// TIA Portal V15.1 export
// export: Created 2024-06-21T08:41:06.8182544Z, ExportSetting WithDefaults, DisplayName Totally Integrated Automation Portal, DisplayVersion V15.1 Update 5, DisplayName TIA Portal Openness, DisplayVersion V15.1 Update 5, DisplayName SINAMICS Startdrive Advanced, DisplayVersion V15.1, DisplayName G130, G150, S120, S150, SINAMICS MV, S210, DisplayVersion V15.1, DisplayName G110M, G120, G120C, G120D, G120P, DisplayVersion V15.1, DisplayName STEP 7 Professional, DisplayVersion V15.1 Update 5, DisplayName STEP 7 Safety, DisplayVersion V15.1, DisplayName WinCC Professional, DisplayVersion V15.1 Update 5, DisplayName SIMATIC Visualization Architect, DisplayVersion V15.1
FUNCTION_BLOCK "LGBProdStartStop"   // FB6645, FBD
TITLE = LGBProdStartStop
{ S7_Optimized_Access := 'TRUE' }
VERSION : 0.1
// stored: AutoNumber false, IsIECCheckEnabled false, IsRetainMemResEnabled false, MemoryReserve 100, SetENOAutomatically False, UDAEnableTagReadback false
   VAR_INPUT
      I_StartReqCR { ExternalAccessible := 'False'; ExternalVisible := 'False'; ExternalWritable := 'False'} : Bool;   // start request by controlroom
      I_StopReqCR { ExternalAccessible := 'False'; ExternalVisible := 'False'; ExternalWritable := 'False'} : Bool;   // stop request by controlroom
      I_StartReqPbLocal { ExternalAccessible := 'False'; ExternalVisible := 'False'; ExternalWritable := 'False'} : Bool;   // start request by local Pushbutton
      I_StopReqPbLocal { ExternalAccessible := 'False'; ExternalVisible := 'False'; ExternalWritable := 'False'} : Bool;   // stop request by local Pushbutton
      I_StopReqInfdWait { ExternalAccessible := 'False'; ExternalVisible := 'False'; ExternalWritable := 'False'} : Bool;   // stop request by infeed Wait state
      I_StopReqOutfdWait { ExternalAccessible := 'False'; ExternalVisible := 'False'; ExternalWritable := 'False'} : Bool;   // stop request by outfeed Wait state
      I_StopReqAndonHcall { ExternalAccessible := 'False'; ExternalVisible := 'False'; ExternalWritable := 'False'} : Bool;   // stop request by Andon - cause H call
      I_StopReqAndonEcall { ExternalAccessible := 'False'; ExternalVisible := 'False'; ExternalWritable := 'False'} : Bool;   // stop request by Andon - cause E call
      I_StopReqAndonMcall { ExternalAccessible := 'False'; ExternalVisible := 'False'; ExternalWritable := 'False'} : Bool;   // stop request by Andon - cause E call
      I_PartsAtFixedLineStop { ExternalAccessible := 'False'; ExternalVisible := 'False'; ExternalWritable := 'False'} : Bool;   // parts are at fixed linstop position (from linefeed module)
      I_SetpCycleTime { ExternalAccessible := 'False'; ExternalVisible := 'False'; ExternalWritable := 'False'} : Int := 60;   // Cycle time (s)
   END_VAR
   VAR_OUTPUT
      O_StartCmd { ExternalAccessible := 'False'; ExternalVisible := 'False'; ExternalWritable := 'False'} : Bool;   // start command to external unit
      O_StopCmd { ExternalAccessible := 'False'; ExternalVisible := 'False'; ExternalWritable := 'False'} : Bool;   // stop command to external unit
      O_IndStart { ExternalAccessible := 'False'; ExternalVisible := 'False'; ExternalWritable := 'False'} : Bool;   // Indication Start for button
      O_IndStop { ExternalAccessible := 'False'; ExternalVisible := 'False'; ExternalWritable := 'False'} : Bool;   // Indication Stop for button
      O_AndonActive { ExternalAccessible := 'False'; ExternalVisible := 'False'; ExternalWritable := 'False'} : Bool;   // andon is active
      O_StoppedByCR { ExternalAccessible := 'False'; ExternalVisible := 'False'; ExternalWritable := 'False'} : Bool;   // state 'stopped by controlroom' is active
      O_StoppedByLocal { ExternalAccessible := 'False'; ExternalVisible := 'False'; ExternalWritable := 'False'} : Bool;   // state 'stopped by local operator action ' is active
      O_StoppedByInfeedWait { ExternalAccessible := 'False'; ExternalVisible := 'False'; ExternalWritable := 'False'} : Bool;   // state 'stopped by infeed wait ' is active
      O_StoppedByOutfeedWait { ExternalAccessible := 'False'; ExternalVisible := 'False'; ExternalWritable := 'False'} : Bool;   // state 'stopped by outfeed wait ' is active
      O_StoppedByAndonHcall { ExternalAccessible := 'False'; ExternalVisible := 'False'; ExternalWritable := 'False'} : Bool;   // stopped by andon H-call
      O_StoppedByAndonEcall { ExternalAccessible := 'False'; ExternalVisible := 'False'; ExternalWritable := 'False'} : Bool;   // stopped by andon E-call
      O_StoppedByAndonMcall { ExternalAccessible := 'False'; ExternalVisible := 'False'; ExternalWritable := 'False'} : Bool;   // stopped by andon E-call
      O_GapsAllowed { ExternalAccessible := 'False'; ExternalVisible := 'False'; ExternalWritable := 'False'} : Bool;   // Gaps Allowed
      O_AlarmABCondition { ExternalAccessible := 'False'; ExternalVisible := 'False'; ExternalWritable := 'False'} : Bool;   // Alarm AB Condition
      O_AlarmA { ExternalAccessible := 'False'; ExternalVisible := 'False'; ExternalWritable := 'False'} : Bool;   // Summation Alarm A of roller. / Alarm A
      O_AlarmB { ExternalAccessible := 'False'; ExternalVisible := 'False'; ExternalWritable := 'False'} : Bool;   // Summation Alarm B of roller. / Alarm B
      O_AlarmC { ExternalAccessible := 'False'; ExternalVisible := 'False'; ExternalWritable := 'False'} : Bool;   // Summation Alarm C of roller. / Alarm C
      O_AlarmD { ExternalAccessible := 'False'; ExternalVisible := 'False'; ExternalWritable := 'False'} : Bool;   // Summation Alarm D of roller. / Alarm D
      H_AlarmDWord { ExternalAccessible := 'False'; ExternalVisible := 'False'; ExternalWritable := 'False'} : DWord;   // Alarm Word
   END_VAR
   VAR_IN_OUT
      IO_Modes : "Modes";   // Modes
      IO_ShiftRegData : "ShiftRegData";   // Line data- from shiftregister
      H_HMI : "H_HMI";   // Animation
      H_GBProdStartStop : "H_GBProdStartStop";   // Animation
      C_Config : "ProdStartStopConfig";   // Config
   END_VAR
   VAR
      AD_StopCR { ExternalAccessible := 'False'; ExternalVisible := 'False'; ExternalWritable := 'False'} : Bool;   // Stop by Control Room
      AD_StopLocal { ExternalAccessible := 'False'; ExternalVisible := 'False'; ExternalWritable := 'False'} : Bool;   // Stop by local stop
      AD_StopAndonHCall { ExternalAccessible := 'False'; ExternalVisible := 'False'; ExternalWritable := 'False'} : Bool;   // Stop by Andon H Call
      AD_StopAndonECall { ExternalAccessible := 'False'; ExternalVisible := 'False'; ExternalWritable := 'False'} : Bool;   // Stop by Andon E Call
      AD_StopAndonMCall { ExternalAccessible := 'False'; ExternalVisible := 'False'; ExternalWritable := 'False'} : Bool;   // Stop by Andon M Call
      AD_AndonNotActive { ExternalAccessible := 'False'; ExternalVisible := 'False'; ExternalWritable := 'False'} : Bool;   // Andon not active
      AD_StopInfeedWait { ExternalAccessible := 'False'; ExternalVisible := 'False'; ExternalWritable := 'False'} : Bool;   // Stop by infeed wait
      AD_StopOutfeedWait { ExternalAccessible := 'False'; ExternalVisible := 'False'; ExternalWritable := 'False'} : Bool;   // Stop by outfeed wait
      AD_GapsAllowed { ExternalAccessible := 'False'; ExternalVisible := 'False'; ExternalWritable := 'False'} : Bool;   // Gaps Allowed
      AndonActive { ExternalAccessible := 'False'; ExternalVisible := 'False'; ExternalWritable := 'False'} : Bool;
      StartReqCRDelayed { ExternalAccessible := 'False'; ExternalVisible := 'False'; ExternalWritable := 'False'} : Bool;
      StopReqCRCond { ExternalAccessible := 'False'; ExternalVisible := 'False'; ExternalWritable := 'False'} : Bool;
      StopReqCRPls { ExternalAccessible := 'False'; ExternalVisible := 'False'; ExternalWritable := 'False'} : Bool;
      StopReqCREdg { ExternalAccessible := 'False'; ExternalVisible := 'False'; ExternalWritable := 'False'} : Bool;
      StopReqCR { ExternalAccessible := 'False'; ExternalVisible := 'False'; ExternalWritable := 'False'} : Bool;
      StopReqCRDelayed { ExternalAccessible := 'False'; ExternalVisible := 'False'; ExternalWritable := 'False'} : Bool;
      StopReqDelayTimerAct { ExternalAccessible := 'False'; ExternalVisible := 'False'; ExternalWritable := 'False'} : DInt;
      StartReqHMIPls { ExternalAccessible := 'False'; ExternalVisible := 'False'; ExternalWritable := 'False'} : Bool;
      StartReqCRPls { ExternalAccessible := 'False'; ExternalVisible := 'False'; ExternalWritable := 'False'} : Bool;
      StartReqCREdg { ExternalAccessible := 'False'; ExternalVisible := 'False'; ExternalWritable := 'False'} : Bool;
      StopReqHMI { ExternalAccessible := 'False'; ExternalVisible := 'False'; ExternalWritable := 'False'} : Bool;
      StopReqAndon { ExternalAccessible := 'False'; ExternalVisible := 'False'; ExternalWritable := 'False'} : Bool;
      StoppedPrepared { ExternalAccessible := 'False'; ExternalVisible := 'False'; ExternalWritable := 'False'} : Bool;
      StartedPrepared { ExternalAccessible := 'False'; ExternalVisible := 'False'; ExternalWritable := 'False'} : Bool;
      StartedPreparedEdge { ExternalAccessible := 'False'; ExternalVisible := 'False'; ExternalWritable := 'False'} : Bool;
      StoppedAtLineOfTime { ExternalAccessible := 'False'; ExternalVisible := 'False'; ExternalWritable := 'False'} : Bool;
      StartReqCRDelayTimerSetp { ExternalAccessible := 'False'; ExternalVisible := 'False'; ExternalWritable := 'False'} : DInt;
      StartReqCRDelayTimerAct { ExternalAccessible := 'False'; ExternalVisible := 'False'; ExternalWritable := 'False'} : DInt;
      StartReqCRDelayTimerActRemain { ExternalAccessible := 'False'; ExternalVisible := 'False'; ExternalWritable := 'False'} : DInt;
      StartReqCRDelayTimerActRemainS { ExternalAccessible := 'False'; ExternalVisible := 'False'; ExternalWritable := 'False'} : DInt;
      StopReqHMIPls { ExternalAccessible := 'False'; ExternalVisible := 'False'; ExternalWritable := 'False'} : Bool;
      StopAndonReqHMIPls { ExternalAccessible := 'False'; ExternalVisible := 'False'; ExternalWritable := 'False'} : Bool;
      StopReqLocalPBEdg { ExternalAccessible := 'False'; ExternalVisible := 'False'; ExternalWritable := 'False'} : Bool;
      StopReqLocalPBPls { ExternalAccessible := 'False'; ExternalVisible := 'False'; ExternalWritable := 'False'} : Bool;
      StartReqLocalPBEdg { ExternalAccessible := 'False'; ExternalVisible := 'False'; ExternalWritable := 'False'} : Bool;
      StartReqLocalPBPls { ExternalAccessible := 'False'; ExternalVisible := 'False'; ExternalWritable := 'False'} : Bool;
      StopReqLocal { ExternalAccessible := 'False'; ExternalVisible := 'False'; ExternalWritable := 'False'} : Bool;
      Stop { ExternalAccessible := 'False'; ExternalVisible := 'False'; ExternalWritable := 'False'} : Bool;
      StoppedbyAndonHCall { ExternalAccessible := 'False'; ExternalVisible := 'False'; ExternalWritable := 'False'} : Bool;
      StoppedbyAndonECall { ExternalAccessible := 'False'; ExternalVisible := 'False'; ExternalWritable := 'False'} : Bool;
      StoppedbyAndonMCall { ExternalAccessible := 'False'; ExternalVisible := 'False'; ExternalWritable := 'False'} : Bool;
   END_VAR
   VAR RETAIN
      GapsAllowed { ExternalAccessible := 'False'; ExternalVisible := 'False'; ExternalWritable := 'False'} : Bool;
   END_VAR
   VAR
      AlarmA { ExternalAccessible := 'False'; ExternalVisible := 'False'; ExternalWritable := 'False'} : Bool;   // Summation Alarm A of roller. / Alarm A
      AlarmB { ExternalAccessible := 'False'; ExternalVisible := 'False'; ExternalWritable := 'False'} : Bool;   // Summation Alarm B of roller. / Alarm B
      AlarmC { ExternalAccessible := 'False'; ExternalVisible := 'False'; ExternalWritable := 'False'} : Bool;   // Summation Alarm C of roller. / Alarm C
      AlarmD { ExternalAccessible := 'False'; ExternalVisible := 'False'; ExternalWritable := 'False'} : Bool;   // Summation Alarm D of roller. / Alarm D
      AlarmABCondition { ExternalAccessible := 'False'; ExternalVisible := 'False'; ExternalWritable := 'False'} : Bool;   // Alarm AB Condition
      CycleTimeSetp { ExternalAccessible := 'False'; ExternalVisible := 'False'; ExternalWritable := 'False'} : DInt;   // cycletime (ms)
      HMICMD { ExternalAccessible := 'False'; ExternalVisible := 'False'; ExternalWritable := 'False'} : Struct   // Temp
         Start { ExternalAccessible := 'False'; ExternalVisible := 'False'; ExternalWritable := 'False'} : Bool;   // Start
         Stop { ExternalAccessible := 'False'; ExternalVisible := 'False'; ExternalWritable := 'False'} : Bool;   // Stop
         StopAndon { ExternalAccessible := 'False'; ExternalVisible := 'False'; ExternalWritable := 'False'} : Bool;   // Stop Andon
         ActivateAndon { ExternalAccessible := 'False'; ExternalVisible := 'False'; ExternalWritable := 'False'} : Bool;   // Activate Andon
         GapsAllowed { ExternalAccessible := 'False'; ExternalVisible := 'False'; ExternalWritable := 'False'} : Bool;   // Gaps Allowed
         Spare5 { ExternalAccessible := 'False'; ExternalVisible := 'False'; ExternalWritable := 'False'} : Bool;   // Spare
         Spare6 { ExternalAccessible := 'False'; ExternalVisible := 'False'; ExternalWritable := 'False'} : Bool;   // Spare
         Spare7 { ExternalAccessible := 'False'; ExternalVisible := 'False'; ExternalWritable := 'False'} : Bool;   // Spare
         Spare8 { ExternalAccessible := 'False'; ExternalVisible := 'False'; ExternalWritable := 'False'} : Bool;   // Spare
         Spare9 { ExternalAccessible := 'False'; ExternalVisible := 'False'; ExternalWritable := 'False'} : Bool;   // Spare
         Spare10 { ExternalAccessible := 'False'; ExternalVisible := 'False'; ExternalWritable := 'False'} : Bool;   // Spare
         Spare11 { ExternalAccessible := 'False'; ExternalVisible := 'False'; ExternalWritable := 'False'} : Bool;   // Spare
         Spare12 { ExternalAccessible := 'False'; ExternalVisible := 'False'; ExternalWritable := 'False'} : Bool;   // Spare
         Spare13 { ExternalAccessible := 'False'; ExternalVisible := 'False'; ExternalWritable := 'False'} : Bool;   // Spare
         Spare14 { ExternalAccessible := 'False'; ExternalVisible := 'False'; ExternalWritable := 'False'} : Bool;   // Spare
         Spare15 { ExternalAccessible := 'False'; ExternalVisible := 'False'; ExternalWritable := 'False'} : Bool;   // Spare
         Spare16 { ExternalAccessible := 'False'; ExternalVisible := 'False'; ExternalWritable := 'False'} : Bool;   // Spare
         Spare17 { ExternalAccessible := 'False'; ExternalVisible := 'False'; ExternalWritable := 'False'} : Bool;   // Spare
         Spare18 { ExternalAccessible := 'False'; ExternalVisible := 'False'; ExternalWritable := 'False'} : Bool;   // Spare
         Spare19 { ExternalAccessible := 'False'; ExternalVisible := 'False'; ExternalWritable := 'False'} : Bool;   // Spare
         Spare20 { ExternalAccessible := 'False'; ExternalVisible := 'False'; ExternalWritable := 'False'} : Bool;   // Spare
         Spare21 { ExternalAccessible := 'False'; ExternalVisible := 'False'; ExternalWritable := 'False'} : Bool;   // Spare
         Spare22 { ExternalAccessible := 'False'; ExternalVisible := 'False'; ExternalWritable := 'False'} : Bool;   // Spare
         Spare23 { ExternalAccessible := 'False'; ExternalVisible := 'False'; ExternalWritable := 'False'} : Bool;   // Spare
         Spare24 { ExternalAccessible := 'False'; ExternalVisible := 'False'; ExternalWritable := 'False'} : Bool;   // Spare
         Spare25 { ExternalAccessible := 'False'; ExternalVisible := 'False'; ExternalWritable := 'False'} : Bool;   // Spare
         Spare26 { ExternalAccessible := 'False'; ExternalVisible := 'False'; ExternalWritable := 'False'} : Bool;   // Spare
         Spare27 { ExternalAccessible := 'False'; ExternalVisible := 'False'; ExternalWritable := 'False'} : Bool;   // Spare
         Spare28 { ExternalAccessible := 'False'; ExternalVisible := 'False'; ExternalWritable := 'False'} : Bool;   // Spare
         Spare29 { ExternalAccessible := 'False'; ExternalVisible := 'False'; ExternalWritable := 'False'} : Bool;   // Spare
         Spare30 { ExternalAccessible := 'False'; ExternalVisible := 'False'; ExternalWritable := 'False'} : Bool;   // Spare
         Spare31 { ExternalAccessible := 'False'; ExternalVisible := 'False'; ExternalWritable := 'False'} : Bool;   // Spare
      END_STRUCT;
      _StartReqCRDelayTimer { ExternalAccessible := 'False'; ExternalVisible := 'False'; ExternalWritable := 'False'} : "LTimer";
      _StopReqCRDelayTimer { ExternalAccessible := 'False'; ExternalVisible := 'False'; ExternalWritable := 'False'} : "LTimer";
      LToggle_GapsAllowed { ExternalAccessible := 'False'; ExternalVisible := 'False'; ExternalWritable := 'False'} : "LToggle";
   END_VAR
   VAR_TEMP   // added for the SCL form of the ladder/FBD networks
      _w1 : Bool;
      _w2 : Bool;
   END_VAR
BEGIN

REGION Network 1: **** 1 - Inputs **** HMI Commands
   // HMI Commands
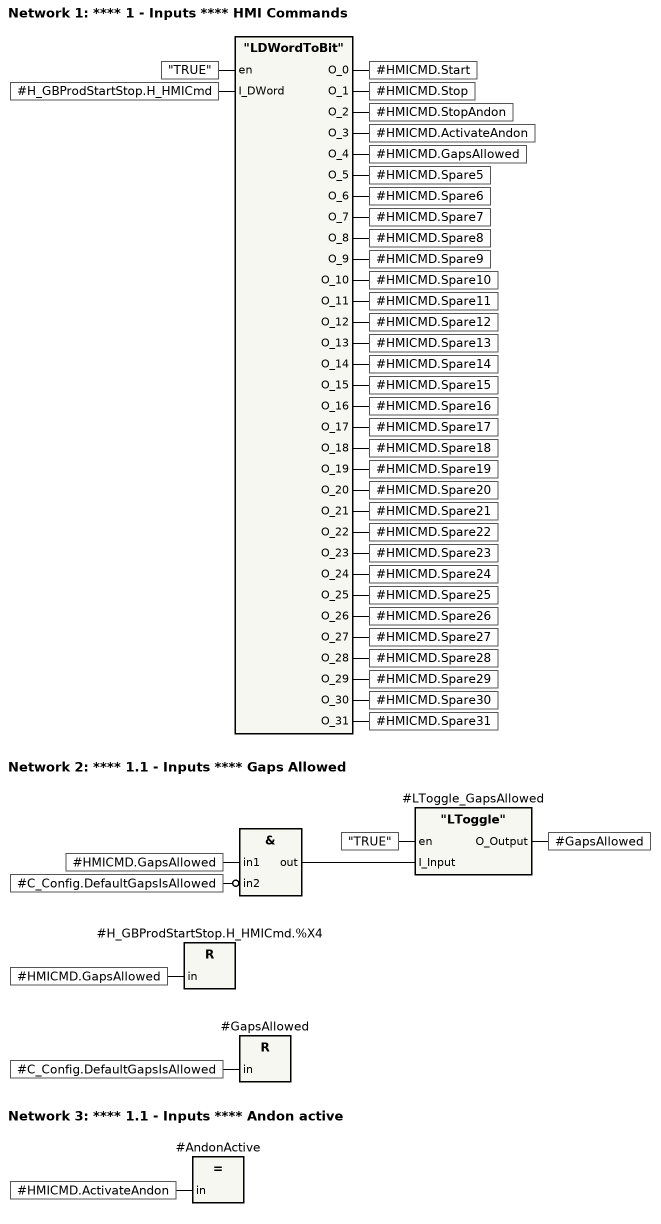
   IF "TRUE" THEN
       "LDWordToBit"(I_DWord := #H_GBProdStartStop.H_HMICmd,
                     O_0 => #HMICMD.Start,
                     O_1 => #HMICMD.Stop,
                     O_2 => #HMICMD.StopAndon,
                     O_3 => #HMICMD.ActivateAndon,
                     O_4 => #HMICMD.GapsAllowed,
                     O_5 => #HMICMD.Spare5,
                     O_6 => #HMICMD.Spare6,
                     O_7 => #HMICMD.Spare7,
                     O_8 => #HMICMD.Spare8,
                     O_9 => #HMICMD.Spare9,
                     O_10 => #HMICMD.Spare10,
                     O_11 => #HMICMD.Spare11,
                     O_12 => #HMICMD.Spare12,
                     O_13 => #HMICMD.Spare13,
                     O_14 => #HMICMD.Spare14,
                     O_15 => #HMICMD.Spare15,
                     O_16 => #HMICMD.Spare16,
                     O_17 => #HMICMD.Spare17,
                     O_18 => #HMICMD.Spare18,
                     O_19 => #HMICMD.Spare19,
                     O_20 => #HMICMD.Spare20,
                     O_21 => #HMICMD.Spare21,
                     O_22 => #HMICMD.Spare22,
                     O_23 => #HMICMD.Spare23,
                     O_24 => #HMICMD.Spare24,
                     O_25 => #HMICMD.Spare25,
                     O_26 => #HMICMD.Spare26,
                     O_27 => #HMICMD.Spare27,
                     O_28 => #HMICMD.Spare28,
                     O_29 => #HMICMD.Spare29,
                     O_30 => #HMICMD.Spare30,
                     O_31 => #HMICMD.Spare31);
   END_IF;
END_REGION

REGION Network 2: **** 1.1 - Inputs **** Gaps Allowed
   IF "TRUE" THEN
       #LToggle_GapsAllowed(I_Input := #HMICMD.GapsAllowed AND NOT #C_Config.DefaultGapsIsAllowed,   // "LToggle"
                            O_Output => #GapsAllowed);
   END_IF;
   IF #HMICMD.GapsAllowed THEN #H_GBProdStartStop.H_HMICmd.%X4 := FALSE; END_IF;
   IF #C_Config.DefaultGapsIsAllowed THEN #GapsAllowed := FALSE; END_IF;
END_REGION

REGION Network 3: **** 1.1 - Inputs **** Andon active
   #AndonActive := #HMICMD.ActivateAndon;
END_REGION

REGION Network 4: **** 1.1 - Inputs **** Pushbutton start request - by HMI - Create pulse
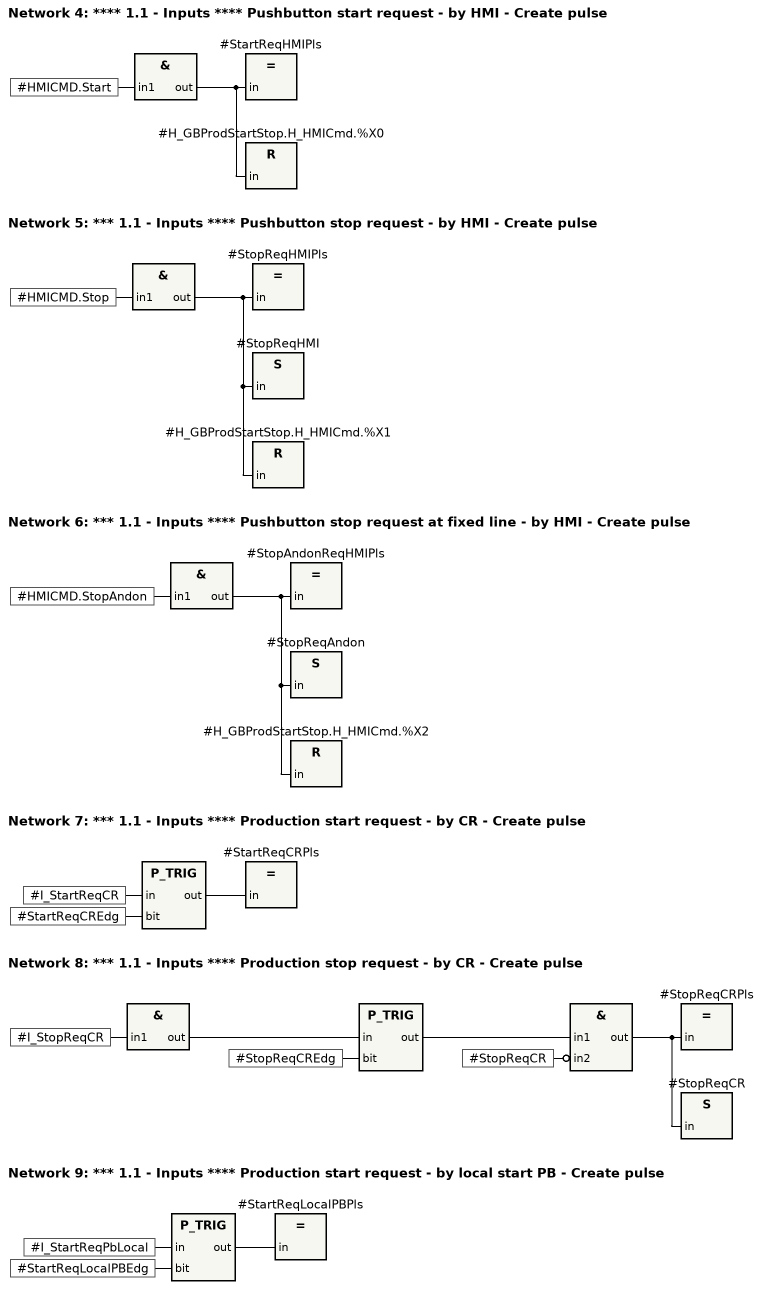
   #StartReqHMIPls := #HMICMD.Start;
   IF #HMICMD.Start THEN #H_GBProdStartStop.H_HMICmd.%X0 := FALSE; END_IF;
END_REGION

REGION Network 5: *** 1.1 - Inputs **** Pushbutton stop request - by HMI - Create pulse
   #StopReqHMIPls := #HMICMD.Stop;
   IF #HMICMD.Stop THEN
       #StopReqHMI := TRUE;
       #H_GBProdStartStop.H_HMICmd.%X1 := FALSE;
   END_IF;
END_REGION

REGION Network 6: *** 1.1 - Inputs **** Pushbutton stop request at fixed line - by HMI - Create pulse
   #StopAndonReqHMIPls := #HMICMD.StopAndon;
   IF #HMICMD.StopAndon THEN
       #StopReqAndon := TRUE;
       #H_GBProdStartStop.H_HMICmd.%X2 := FALSE;
   END_IF;
END_REGION

REGION Network 7: *** 1.1 - Inputs **** Production start request - by CR - Create pulse
   #_w1 := #I_StartReqCR AND NOT #StartReqCREdg;   // rising edge
   #StartReqCREdg := #I_StartReqCR;
   #StartReqCRPls := #_w1;
END_REGION

REGION Network 8: *** 1.1 - Inputs **** Production stop request - by CR - Create pulse
   #_w1 := #I_StopReqCR AND NOT #StopReqCREdg;   // rising edge
   #StopReqCREdg := #I_StopReqCR;
   #StopReqCRPls := #_w1 AND NOT #StopReqCR;
   IF #StopReqCRPls THEN #StopReqCR := TRUE; END_IF;
END_REGION

REGION Network 9: *** 1.1 - Inputs **** Production start request - by local start PB - Create pulse
   #_w1 := #I_StartReqPbLocal AND NOT #StartReqLocalPBEdg;   // rising edge
   #StartReqLocalPBEdg := #I_StartReqPbLocal;
   #StartReqLocalPBPls := #_w1;
END_REGION

REGION Network 10: *** 1.1 - Inputs **** Production stop request - by local stop PB - Create pulse
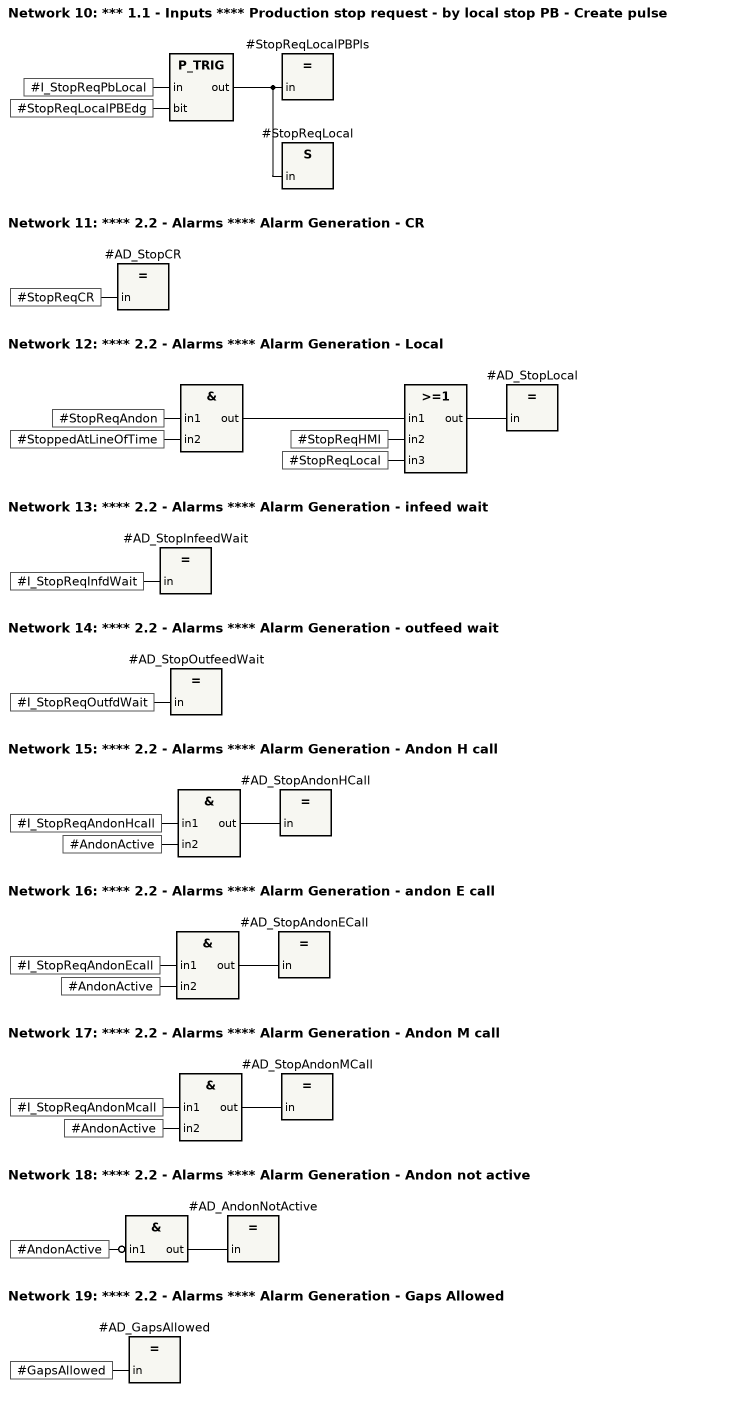
   #_w1 := #I_StopReqPbLocal AND NOT #StopReqLocalPBEdg;   // rising edge
   #StopReqLocalPBEdg := #I_StopReqPbLocal;
   #StopReqLocalPBPls := #_w1;
   IF #_w1 THEN #StopReqLocal := TRUE; END_IF;
END_REGION

REGION Network 11: **** 2.2 - Alarms **** Alarm Generation - CR
   #AD_StopCR := #StopReqCR;
END_REGION

REGION Network 12: **** 2.2 - Alarms **** Alarm Generation - Local
   #AD_StopLocal := (#StopReqAndon AND #StoppedAtLineOfTime) OR #StopReqHMI OR #StopReqLocal;
END_REGION

REGION Network 13: **** 2.2 - Alarms **** Alarm Generation - infeed wait
   #AD_StopInfeedWait := #I_StopReqInfdWait;
END_REGION

REGION Network 14: **** 2.2 - Alarms **** Alarm Generation - outfeed wait
   #AD_StopOutfeedWait := #I_StopReqOutfdWait;
END_REGION

REGION Network 15: **** 2.2 - Alarms **** Alarm Generation - Andon H call
   #AD_StopAndonHCall := #I_StopReqAndonHcall AND #AndonActive;
END_REGION

REGION Network 16: **** 2.2 - Alarms **** Alarm Generation - andon E call
   #AD_StopAndonECall := #I_StopReqAndonEcall AND #AndonActive;
END_REGION

REGION Network 17: **** 2.2 - Alarms **** Alarm Generation - Andon M call
   #AD_StopAndonMCall := #I_StopReqAndonMcall AND #AndonActive;
END_REGION

REGION Network 18: **** 2.2 - Alarms **** Alarm Generation - Andon not active
   #AD_AndonNotActive := NOT #AndonActive;
END_REGION

REGION Network 19: **** 2.2 - Alarms **** Alarm Generation - Gaps Allowed
   #AD_GapsAllowed := #GapsAllowed;
END_REGION

REGION Network 20: *** 4.6 - Machine Status - Indication **** Icon Animation
   // Icon Animation
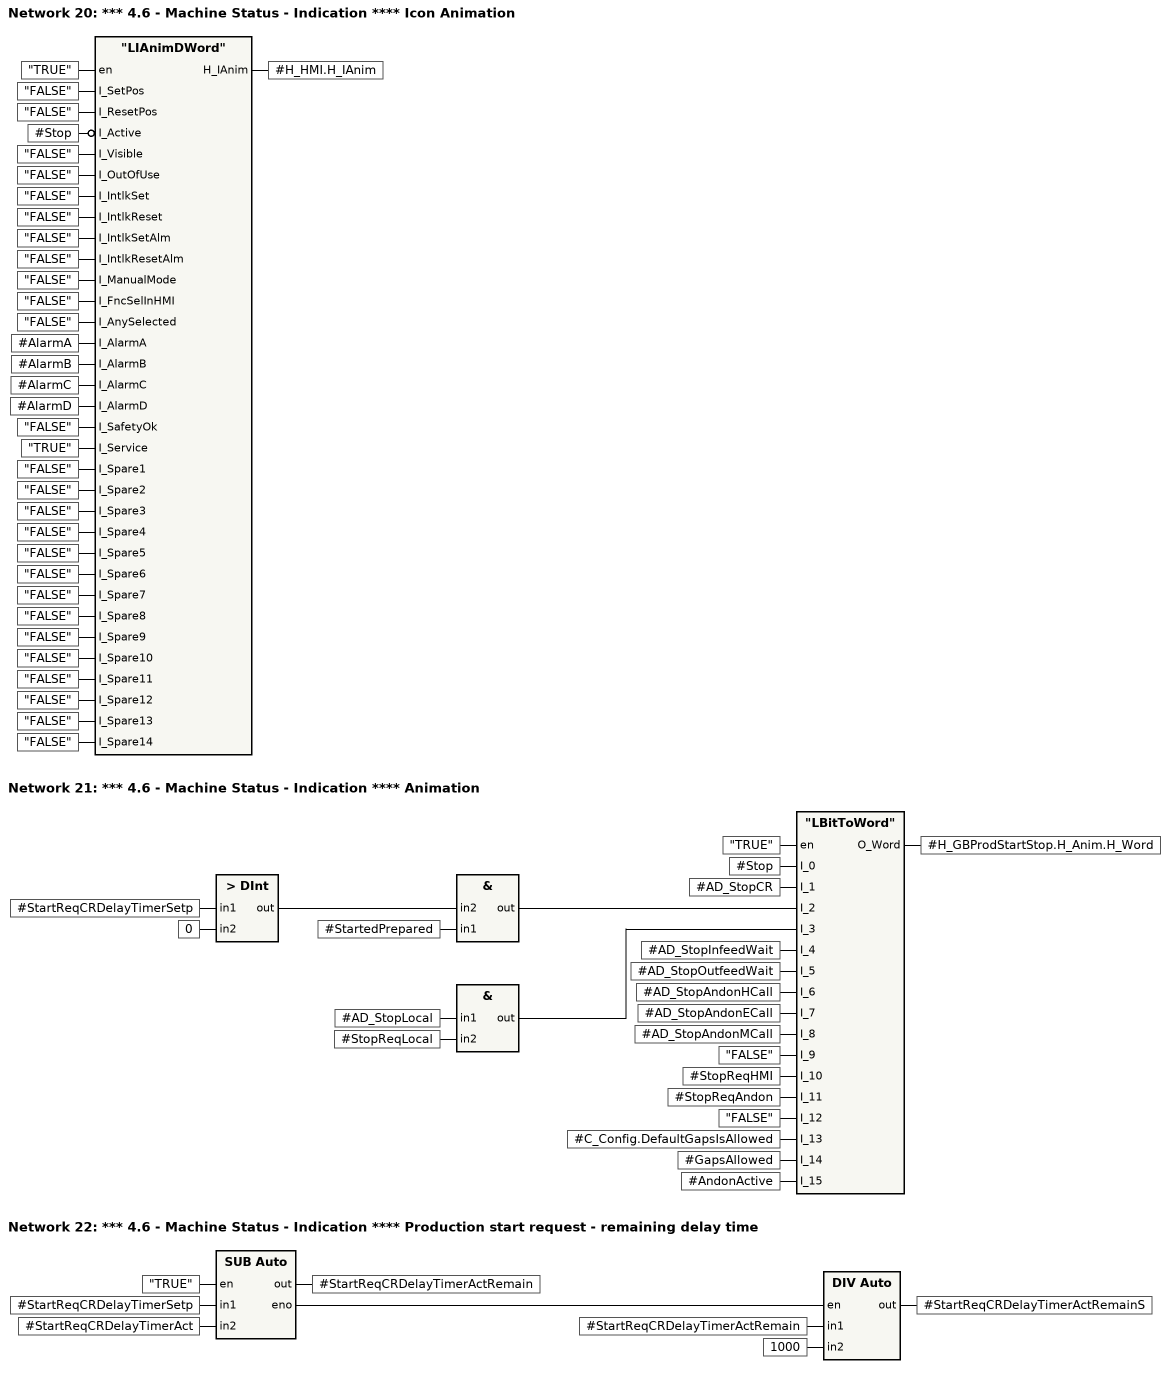
   IF "TRUE" THEN
       "LIAnimDWord"(I_SetPos := "FALSE",
                     I_ResetPos := "FALSE",
                     I_Active := NOT #Stop,
                     I_Visible := "FALSE",
                     I_OutOfUse := "FALSE",
                     I_IntlkSet := "FALSE",
                     I_IntlkReset := "FALSE",
                     I_IntlkSetAlm := "FALSE",
                     I_IntlkResetAlm := "FALSE",
                     I_ManualMode := "FALSE",
                     I_FncSelInHMI := "FALSE",
                     I_AnySelected := "FALSE",
                     I_AlarmA := #AlarmA,
                     I_AlarmB := #AlarmB,
                     I_AlarmC := #AlarmC,
                     I_AlarmD := #AlarmD,
                     I_SafetyOk := "FALSE",
                     I_Service := "TRUE",
                     I_Spare1 := "FALSE",
                     I_Spare2 := "FALSE",
                     I_Spare3 := "FALSE",
                     I_Spare4 := "FALSE",
                     I_Spare5 := "FALSE",
                     I_Spare6 := "FALSE",
                     I_Spare7 := "FALSE",
                     I_Spare8 := "FALSE",
                     I_Spare9 := "FALSE",
                     I_Spare10 := "FALSE",
                     I_Spare11 := "FALSE",
                     I_Spare12 := "FALSE",
                     I_Spare13 := "FALSE",
                     I_Spare14 := "FALSE",
                     H_IAnim => #H_HMI.H_IAnim);
   END_IF;
END_REGION

REGION Network 21: *** 4.6 - Machine Status - Indication **** Animation
   IF "TRUE" THEN
       "LBitToWord"(I_0 := #Stop,
                    I_1 := #AD_StopCR,
                    I_2 := (#StartReqCRDelayTimerSetp > 0) AND #StartedPrepared,
                    I_3 := #AD_StopLocal AND #StopReqLocal,
                    I_4 := #AD_StopInfeedWait,
                    I_5 := #AD_StopOutfeedWait,
                    I_6 := #AD_StopAndonHCall,
                    I_7 := #AD_StopAndonECall,
                    I_8 := #AD_StopAndonMCall,
                    I_9 := "FALSE",
                    I_10 := #StopReqHMI,
                    I_11 := #StopReqAndon,
                    I_12 := "FALSE",
                    I_13 := #C_Config.DefaultGapsIsAllowed,
                    I_14 := #GapsAllowed,
                    I_15 := #AndonActive,
                    O_Word => #H_GBProdStartStop.H_Anim.H_Word);
   END_IF;
END_REGION

REGION Network 22: *** 4.6 - Machine Status - Indication **** Production start request - remaining delay time
   IF "TRUE" THEN
       #StartReqCRDelayTimerActRemain := #StartReqCRDelayTimerSetp - #StartReqCRDelayTimerAct;
       #StartReqCRDelayTimerActRemainS := #StartReqCRDelayTimerActRemain / 1000;
   END_IF;
END_REGION

REGION Network 23: *** 4.6 - Machine Status - Indication **** Wait time start
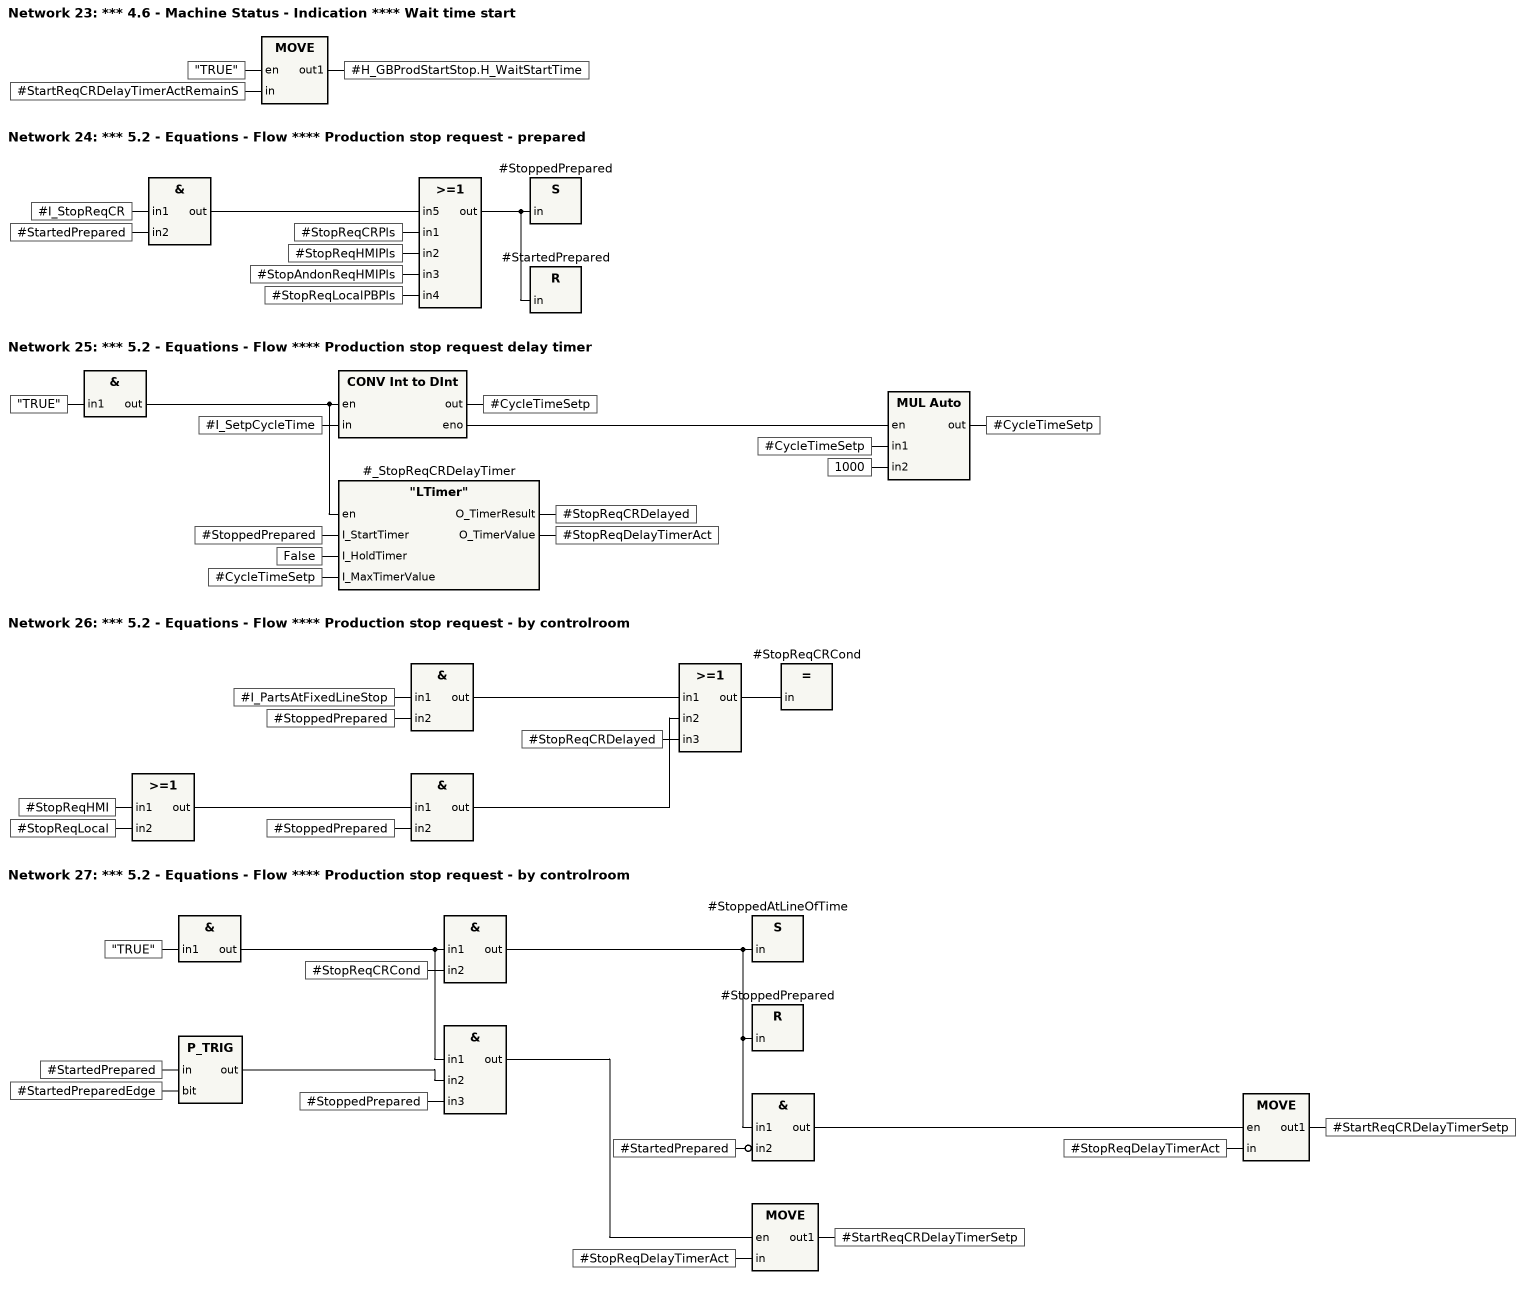
   IF "TRUE" THEN #H_GBProdStartStop.H_WaitStartTime := #StartReqCRDelayTimerActRemainS; END_IF;
END_REGION

REGION Network 24: *** 5.2 - Equations - Flow **** Production stop request - prepared
   IF (#I_StopReqCR AND #StartedPrepared) OR #StopReqCRPls OR #StopReqHMIPls OR #StopAndonReqHMIPls OR #StopReqLocalPBPls THEN
       #StoppedPrepared := TRUE;
       #StartedPrepared := FALSE;
   END_IF;
END_REGION

REGION Network 25: *** 5.2 - Equations - Flow **** Production stop request delay timer
   IF "TRUE" THEN
       #CycleTimeSetp := INT_TO_DINT(#I_SetpCycleTime);
       #CycleTimeSetp := #CycleTimeSetp * 1000;
       #_StopReqCRDelayTimer(I_StartTimer := #StoppedPrepared,   // "LTimer"
                             I_HoldTimer := False,
                             I_MaxTimerValue := #CycleTimeSetp,
                             O_TimerResult => #StopReqCRDelayed,
                             O_TimerValue => #StopReqDelayTimerAct);
   END_IF;
END_REGION

REGION Network 26: *** 5.2 - Equations - Flow **** Production stop request - by controlroom
   #StopReqCRCond := (#I_PartsAtFixedLineStop AND #StoppedPrepared) OR ((#StopReqHMI OR #StopReqLocal) AND #StoppedPrepared) OR #StopReqCRDelayed;
END_REGION

REGION Network 27: *** 5.2 - Equations - Flow **** Production stop request - by controlroom
   #_w1 := "TRUE" AND #StopReqCRCond;
   IF #_w1 THEN
       #StoppedAtLineOfTime := TRUE;
       #StoppedPrepared := FALSE;
   END_IF;
   IF #_w1 AND NOT #StartedPrepared THEN #StartReqCRDelayTimerSetp := #StopReqDelayTimerAct; END_IF;
   #_w2 := #StartedPrepared AND NOT #StartedPreparedEdge;   // rising edge
   #StartedPreparedEdge := #StartedPrepared;
   IF "TRUE" AND #_w2 AND #StoppedPrepared THEN #StartReqCRDelayTimerSetp := #StopReqDelayTimerAct; END_IF;
END_REGION

REGION Network 28: *** 5.2 - Equations - Flow **** Production start request - prepared
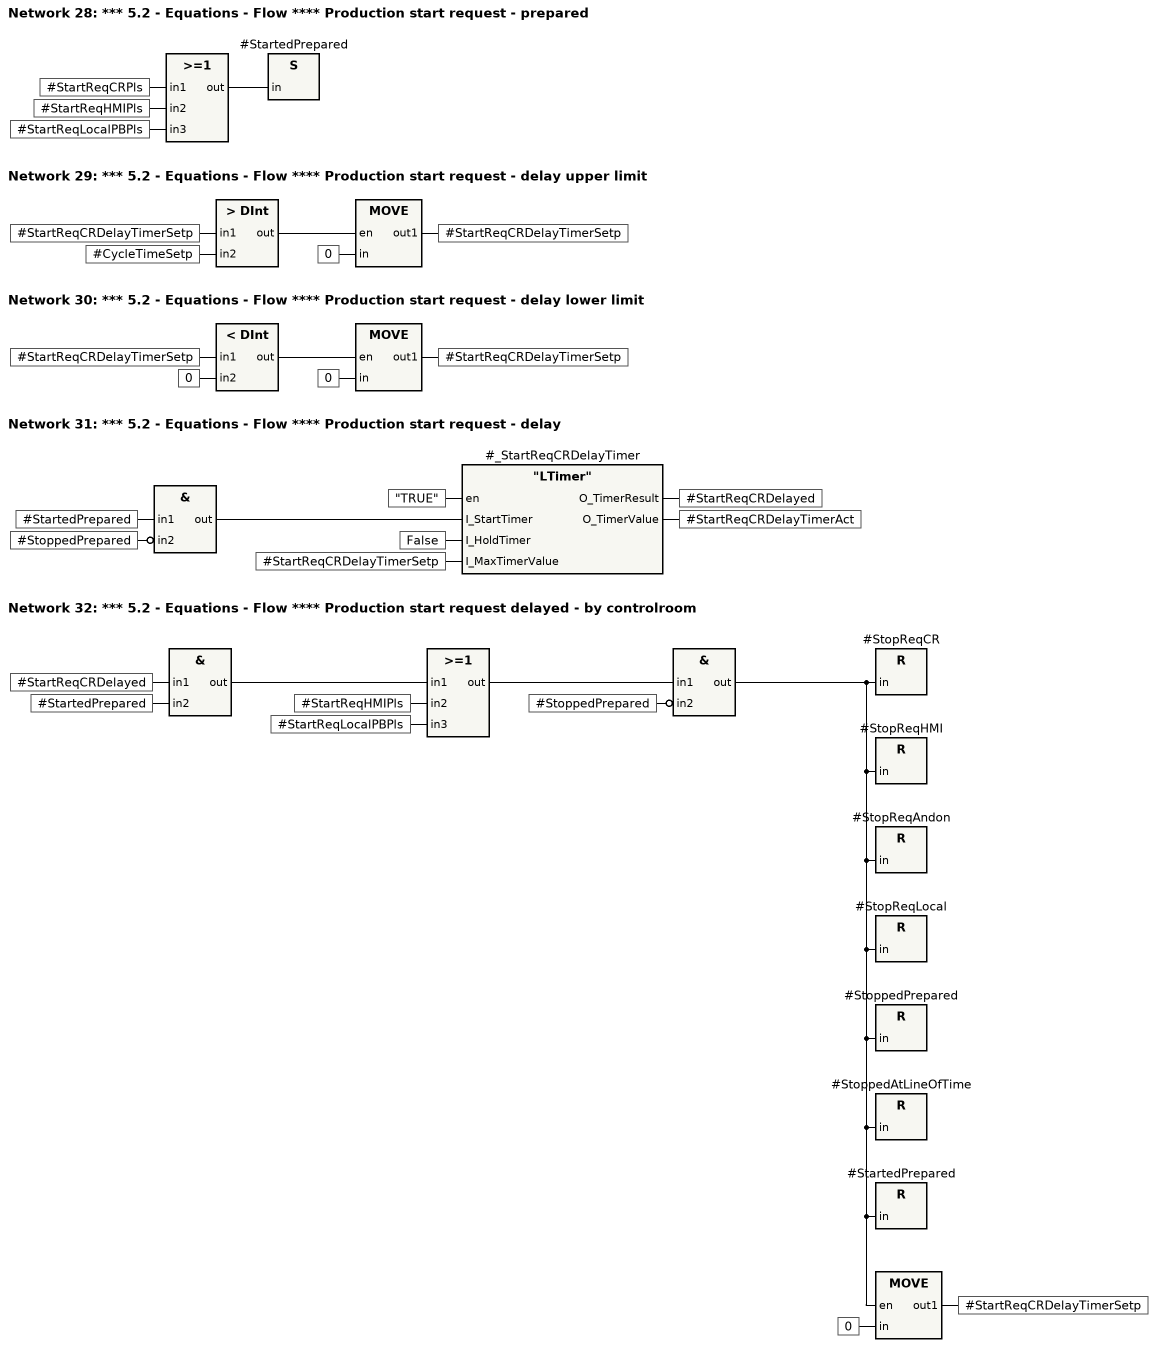
   IF #StartReqCRPls OR #StartReqHMIPls OR #StartReqLocalPBPls THEN #StartedPrepared := TRUE; END_IF;
END_REGION

REGION Network 29: *** 5.2 - Equations - Flow **** Production start request - delay upper limit
   IF #StartReqCRDelayTimerSetp > #CycleTimeSetp THEN #StartReqCRDelayTimerSetp := 0; END_IF;
END_REGION

REGION Network 30: *** 5.2 - Equations - Flow **** Production start request - delay lower limit
   IF #StartReqCRDelayTimerSetp < 0 THEN #StartReqCRDelayTimerSetp := 0; END_IF;
END_REGION

REGION Network 31: *** 5.2 - Equations - Flow **** Production start request - delay
   IF "TRUE" THEN
       #_StartReqCRDelayTimer(I_StartTimer := #StartedPrepared AND NOT #StoppedPrepared,   // "LTimer"
                              I_HoldTimer := False,
                              I_MaxTimerValue := #StartReqCRDelayTimerSetp,
                              O_TimerResult => #StartReqCRDelayed,
                              O_TimerValue => #StartReqCRDelayTimerAct);
   END_IF;
END_REGION

REGION Network 32: *** 5.2 - Equations - Flow **** Production start request delayed - by controlroom
   IF ((#StartReqCRDelayed AND #StartedPrepared) OR #StartReqHMIPls OR #StartReqLocalPBPls) AND NOT #StoppedPrepared THEN
       #StopReqCR := FALSE;
       #StopReqHMI := FALSE;
       #StopReqAndon := FALSE;
       #StopReqLocal := FALSE;
   END_IF;
   #_w1 := ((#StartReqCRDelayed AND #StartedPrepared) OR #StartReqHMIPls OR #StartReqLocalPBPls) AND NOT #StoppedPrepared;
   IF #_w1 THEN
       #StoppedPrepared := FALSE;
       #StoppedAtLineOfTime := FALSE;
       #StartedPrepared := FALSE;
       #StartReqCRDelayTimerSetp := 0;
   END_IF;
END_REGION

REGION Network 33: *** 5.2 - Equations - Flow **** stopped at line of time
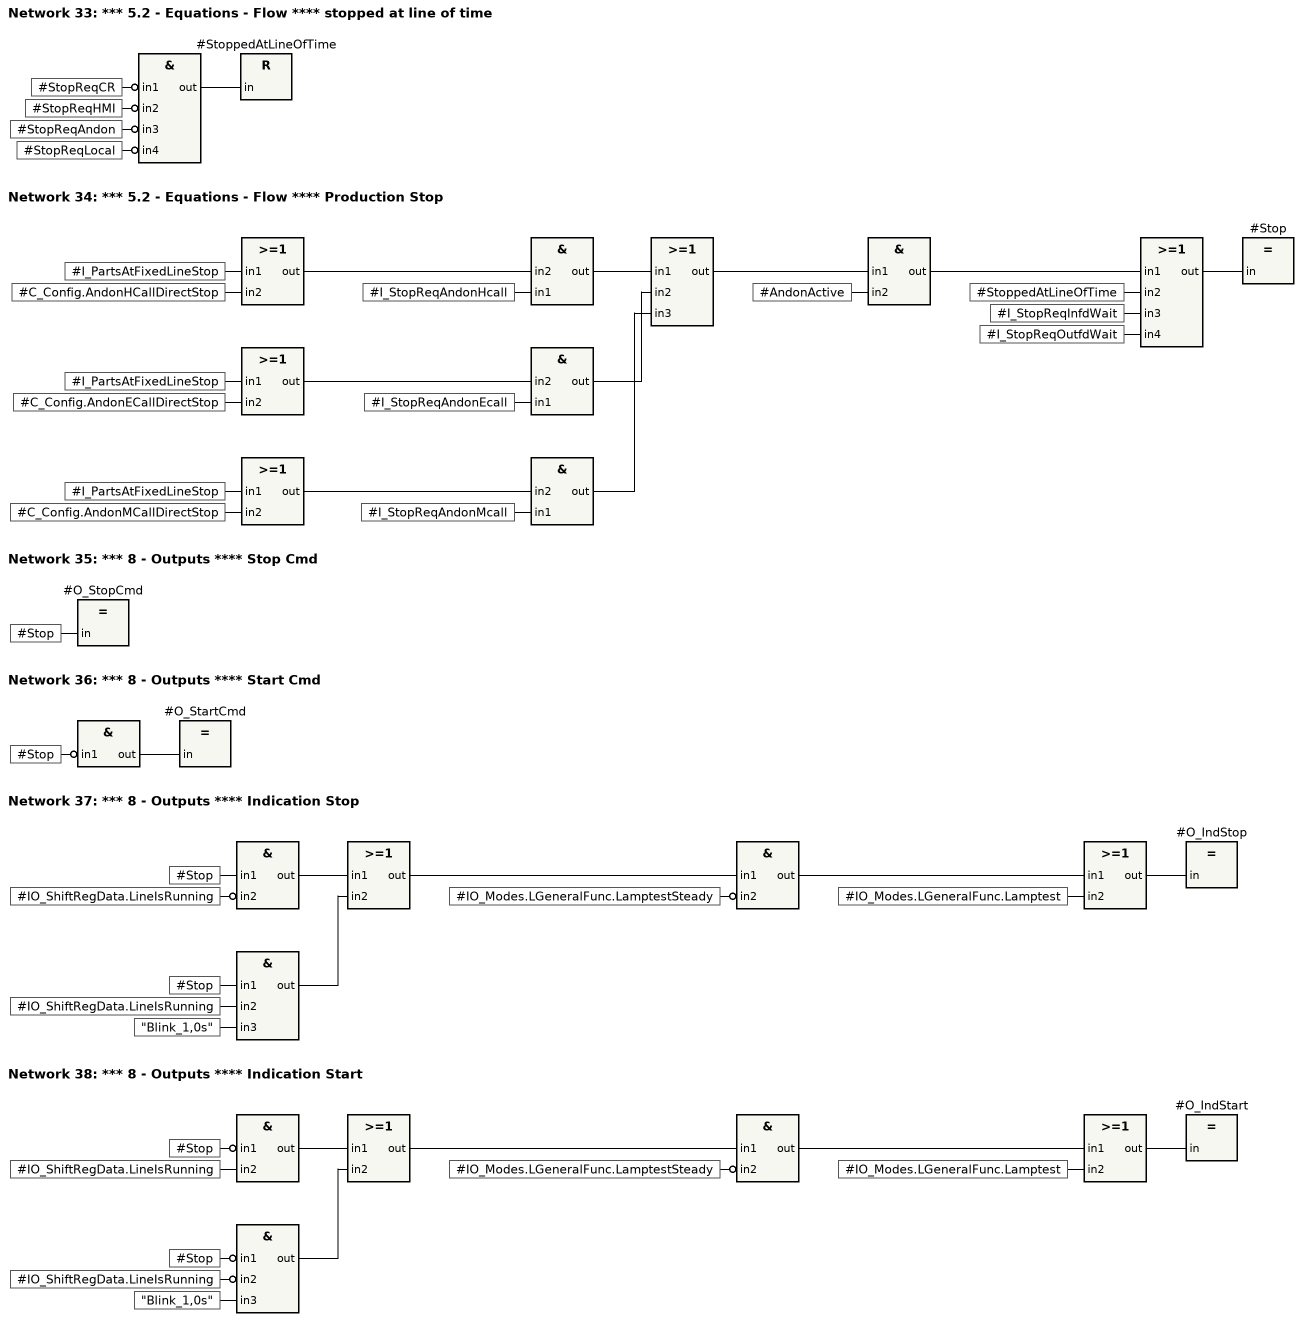
   IF NOT #StopReqCR AND NOT #StopReqHMI AND NOT #StopReqAndon AND NOT #StopReqLocal THEN
       #StoppedAtLineOfTime := FALSE;
   END_IF;
END_REGION

REGION Network 34: *** 5.2 - Equations - Flow **** Production Stop
   #Stop := ((((#I_PartsAtFixedLineStop OR #C_Config.AndonHCallDirectStop) AND #I_StopReqAndonHcall) OR ((#I_PartsAtFixedLineStop OR #C_Config.AndonECallDirectStop) AND #I_StopReqAndonEcall) OR ((#I_PartsAtFixedLineStop OR #C_Config.AndonMCallDirectStop) AND #I_StopReqAndonMcall)) AND #AndonActive) OR #StoppedAtLineOfTime OR #I_StopReqInfdWait OR #I_StopReqOutfdWait;
END_REGION

REGION Network 35: *** 8 - Outputs **** Stop Cmd
   #O_StopCmd := #Stop;
END_REGION

REGION Network 36: *** 8 - Outputs **** Start Cmd
   #O_StartCmd := NOT #Stop;
END_REGION

REGION Network 37: *** 8 - Outputs **** Indication Stop
   #O_IndStop := (((#Stop AND NOT #IO_ShiftRegData.LineIsRunning) OR (#Stop AND #IO_ShiftRegData.LineIsRunning AND "Blink_1,0s")) AND NOT #IO_Modes.LGeneralFunc.LamptestSteady) OR #IO_Modes.LGeneralFunc.Lamptest;
END_REGION

REGION Network 38: *** 8 - Outputs **** Indication Start
   #O_IndStart := (((NOT #Stop AND #IO_ShiftRegData.LineIsRunning) OR (NOT #Stop AND NOT #IO_ShiftRegData.LineIsRunning AND "Blink_1,0s")) AND NOT #IO_Modes.LGeneralFunc.LamptestSteady) OR #IO_Modes.LGeneralFunc.Lamptest;
END_REGION

REGION Network 39: *** 8 - Outputs **** Andon active
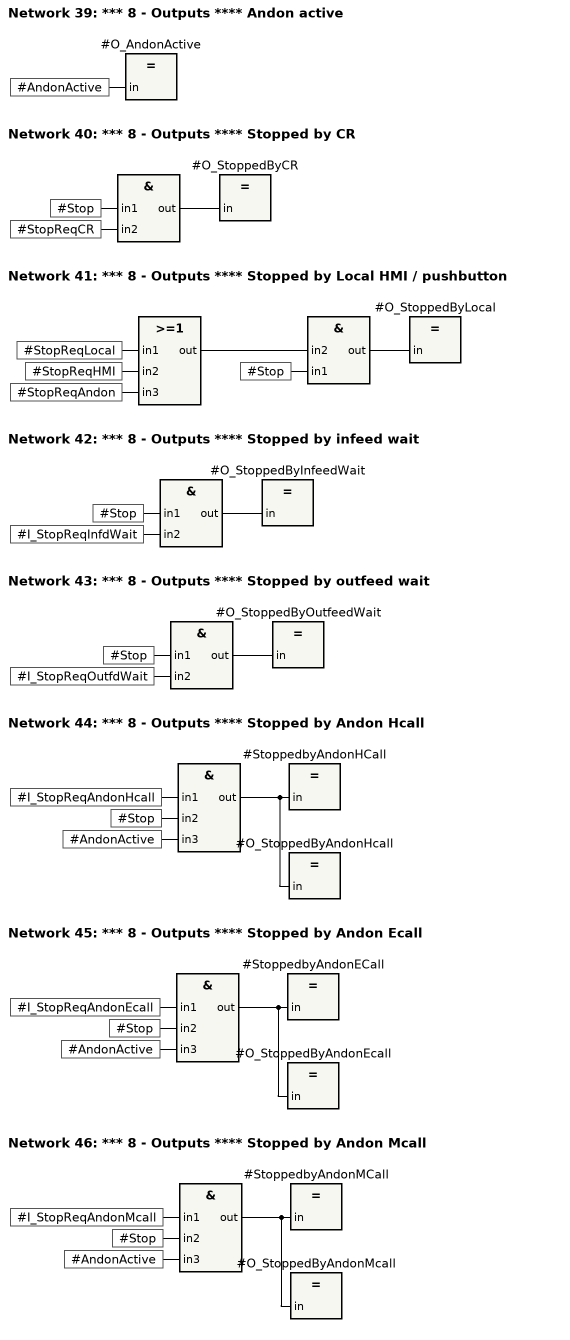
   #O_AndonActive := #AndonActive;
END_REGION

REGION Network 40: *** 8 - Outputs **** Stopped by CR
   #O_StoppedByCR := #Stop AND #StopReqCR;
END_REGION

REGION Network 41: *** 8 - Outputs **** Stopped by Local HMI / pushbutton
   #O_StoppedByLocal := (#StopReqLocal OR #StopReqHMI OR #StopReqAndon) AND #Stop;
END_REGION

REGION Network 42: *** 8 - Outputs **** Stopped by infeed wait
   #O_StoppedByInfeedWait := #Stop AND #I_StopReqInfdWait;
END_REGION

REGION Network 43: *** 8 - Outputs **** Stopped by outfeed wait
   #O_StoppedByOutfeedWait := #Stop AND #I_StopReqOutfdWait;
END_REGION

REGION Network 44: *** 8 - Outputs **** Stopped by Andon Hcall
   #StoppedbyAndonHCall := #I_StopReqAndonHcall AND #Stop AND #AndonActive;
   #O_StoppedByAndonHcall := #StoppedbyAndonHCall;
END_REGION

REGION Network 45: *** 8 - Outputs **** Stopped by Andon Ecall
   #StoppedbyAndonECall := #I_StopReqAndonEcall AND #Stop AND #AndonActive;
   #O_StoppedByAndonEcall := #StoppedbyAndonECall;
END_REGION

REGION Network 46: *** 8 - Outputs **** Stopped by Andon Mcall
   #StoppedbyAndonMCall := #I_StopReqAndonMcall AND #Stop AND #AndonActive;
   #O_StoppedByAndonMcall := #StoppedbyAndonMCall;
END_REGION

REGION Network 47: *** 8 - Outputs **** Gaps Allowed
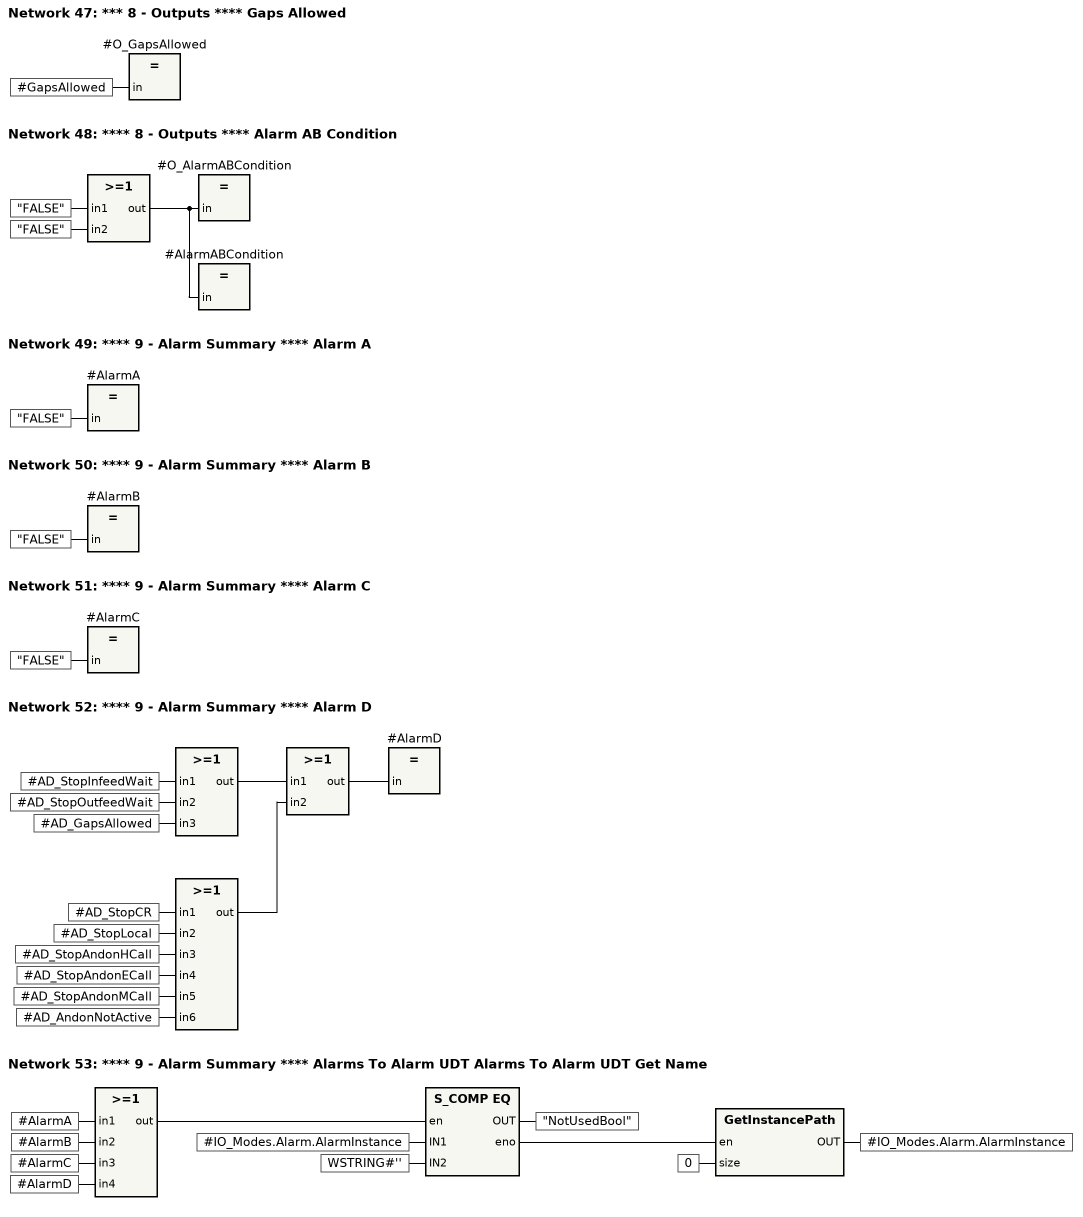
   #O_GapsAllowed := #GapsAllowed;
END_REGION

REGION Network 48: **** 8 - Outputs **** Alarm AB Condition
   // Alarm AB Condition
   #O_AlarmABCondition := "FALSE" OR "FALSE";
   #AlarmABCondition := #O_AlarmABCondition;
END_REGION

REGION Network 49: **** 9 - Alarm Summary **** Alarm A
   // Alarm A
   #AlarmA := "FALSE";
END_REGION

REGION Network 50: **** 9 - Alarm Summary **** Alarm B
   // Alarm B
   #AlarmB := "FALSE";
END_REGION

REGION Network 51: **** 9 - Alarm Summary **** Alarm C
   // Alarm C
   #AlarmC := "FALSE";
END_REGION

REGION Network 52: **** 9 - Alarm Summary **** Alarm D
   // Alarm D
   #AlarmD := #AD_StopInfeedWait OR #AD_StopOutfeedWait OR #AD_GapsAllowed OR #AD_StopCR OR #AD_StopLocal OR #AD_StopAndonHCall OR #AD_StopAndonECall OR #AD_StopAndonMCall OR #AD_AndonNotActive;
END_REGION

REGION Network 53: **** 9 - Alarm Summary **** Alarms To Alarm UDT Alarms To Alarm UDT Get Name
   // Alarm / Alarm D
   S_COMP(EN := #AlarmA OR #AlarmB OR #AlarmC OR #AlarmD,
          IN1 := #IO_Modes.Alarm.AlarmInstance,
          IN2 := WSTRING#'',
          OUT => "NotUsedBool",
          ENO => #_w1);
   IF #_w1 THEN GetInstancePath(size := 0, OUT => #IO_Modes.Alarm.AlarmInstance); END_IF;
END_REGION

REGION Network 54: **** 9 - Alarm Summary **** Alarms To Alarm UDT
   // Alarm / Alarm D
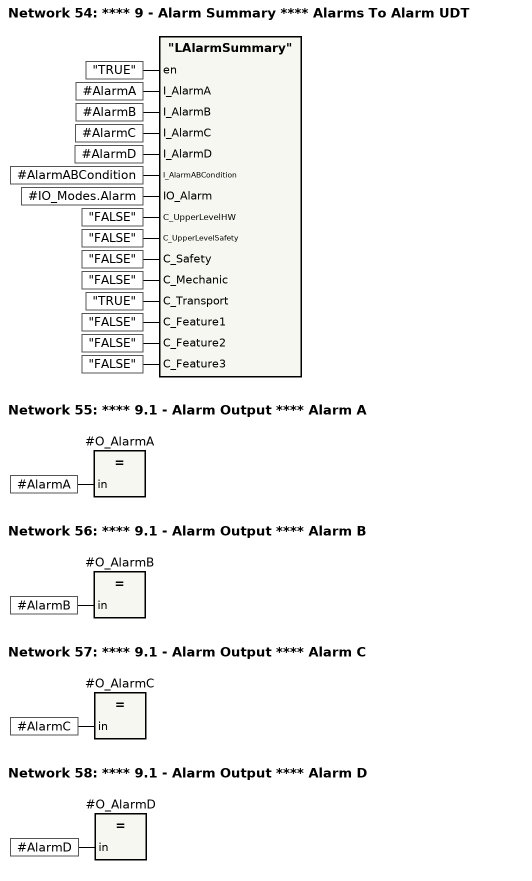
   IF "TRUE" THEN
       "LAlarmSummary"(I_AlarmA := #AlarmA,
                       I_AlarmB := #AlarmB,
                       I_AlarmC := #AlarmC,
                       I_AlarmD := #AlarmD,
                       I_AlarmABCondition := #AlarmABCondition,
                       IO_Alarm := #IO_Modes.Alarm,
                       C_UpperLevelHW := "FALSE",
                       C_UpperLevelSafety := "FALSE",
                       C_Safety := "FALSE",
                       C_Mechanic := "FALSE",
                       C_Transport := "TRUE",
                       C_Feature1 := "FALSE",
                       C_Feature2 := "FALSE",
                       C_Feature3 := "FALSE");
   END_IF;
END_REGION

REGION Network 55: **** 9.1 - Alarm Output **** Alarm A
   // Alarm A
   #O_AlarmA := #AlarmA;
END_REGION

REGION Network 56: **** 9.1 - Alarm Output **** Alarm B
   // Alarm B
   #O_AlarmB := #AlarmB;
END_REGION

REGION Network 57: **** 9.1 - Alarm Output **** Alarm C
   // Alarm C
   #O_AlarmC := #AlarmC;
END_REGION

REGION Network 58: **** 9.1 - Alarm Output **** Alarm D
   // Alarm D
   #O_AlarmD := #AlarmD;
END_REGION

REGION Network 59: **** 9.2 - Alarm DWord**** Alarm To DWord
   // Alarm To Word
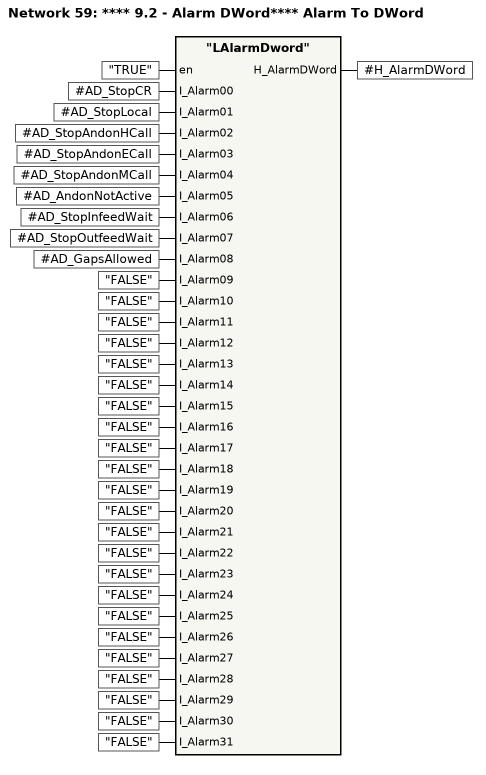
   IF "TRUE" THEN
       "LAlarmDword"(I_Alarm00 := #AD_StopCR,
                     I_Alarm01 := #AD_StopLocal,
                     I_Alarm02 := #AD_StopAndonHCall,
                     I_Alarm03 := #AD_StopAndonECall,
                     I_Alarm04 := #AD_StopAndonMCall,
                     I_Alarm05 := #AD_AndonNotActive,
                     I_Alarm06 := #AD_StopInfeedWait,
                     I_Alarm07 := #AD_StopOutfeedWait,
                     I_Alarm08 := #AD_GapsAllowed,
                     I_Alarm09 := "FALSE",
                     I_Alarm10 := "FALSE",
                     I_Alarm11 := "FALSE",
                     I_Alarm12 := "FALSE",
                     I_Alarm13 := "FALSE",
                     I_Alarm14 := "FALSE",
                     I_Alarm15 := "FALSE",
                     I_Alarm16 := "FALSE",
                     I_Alarm17 := "FALSE",
                     I_Alarm18 := "FALSE",
                     I_Alarm19 := "FALSE",
                     I_Alarm20 := "FALSE",
                     I_Alarm21 := "FALSE",
                     I_Alarm22 := "FALSE",
                     I_Alarm23 := "FALSE",
                     I_Alarm24 := "FALSE",
                     I_Alarm25 := "FALSE",
                     I_Alarm26 := "FALSE",
                     I_Alarm27 := "FALSE",
                     I_Alarm28 := "FALSE",
                     I_Alarm29 := "FALSE",
                     I_Alarm30 := "FALSE",
                     I_Alarm31 := "FALSE",
                     H_AlarmDWord => #H_AlarmDWord);
   END_IF;
END_REGION
END_FUNCTION_BLOCK
